(* Logix 5000 project; controller WWTP_SOLIDS_CLX vendor 1 type 14 code 54 rev 17.2; software revision 17.00; part 11 of 16 *)

ADD_ON_INSTRUCTION P_ResInh   (* revision 0.12, ExecutePrescan, ExecuteEnableInFalse *)
// Restart Inhibit
// Revision note:
// Aligned name, description and local STRING values, sizes, across instructions.
// Help:
// This Instruction monitors starts, running and stops of a motor and decides, based
// on rules for winding heating, when the motor can be started again.
// This Instruction uses a state model, which is documented in the User
// Documentation for the instruction.  It has the following states:
// *  S01:  Cold Motor Ready to Start
// *  S02:  Cold Motor Starting
// *  S03:  Cold Motor Running
// *  S04:  Cold Motor First Failure to Start
// *  S05:  Cold Motor Subsequent Failure to Start
// *  S06:  Hot Motor Starting
// *  S07:  Hot Motor Running
// *  S08:  Hot Motor Short Run Then Stopped
// *  S09:  Hot Motor Long Run Then Stopped
// *  S10:  Hot Motor First Failure to Start
// *  S11:  Hot Motor Subsequent Failure to Start
// *  S12:  Hot Motor Ready to Start
// NOTE:  This is a very basic state model for motor heating and is not intended
// as a close physical model of any given motor.  It cannot replace more
// extensive or sensor-based motor monitoring and modelling systems.
// NOTE:  EnableInFalse (false rung) is treated the same a motor stopped
// (Inp_Starting = 0, Inp_Running = 0, Inp_Stopped = 1).
VAR_INPUT
   Inp_Stopped : BOOL; {visible}   // Equipment is confirmed Stopped
   Inp_Starting : BOOL; {visible}   // Equipment is Starting, indicating a start attempt
   Inp_Running : BOOL := 1; {visible}   // Equipment is confirmed Running
   Cfg_ThreeColdStarts : DINT := 1800;   // Sec within which three starts are allowed if cold
   Cfg_FirstFailCold : DINT := 1800;   // Sec for cold motor to wait after 1st start failure before ready to start
   Cfg_SubseqFailCold : DINT := 14400;   // Sec for cold motor to wait after 2nd and subsequent start failure before ready
   Cfg_FirstFailHot : DINT := 1800;   // Sec for hot motor to wait after 1st start failure before ready to start
   Cfg_SubseqFailHot : DINT := 14400;   // Sec for hot motor to wait after 2nd and subsequent start failure before ready
   Cfg_HotRestartOK : DINT := 3600;   // Sec for hot motor to run so it can immediately restart after stop
   Cfg_RestartHot : DINT := 3600;   // Sec for hot motor to wait after stop if stopped before Hot Restart OK time
   Cfg_HotToCold : DINT := 57600;   // Sec for a stopped hot motor to become cold
END_VAR
VAR_OUTPUT
   Val_MinToReady : DINT; {visible}   // Minutes yet inhibited before ready to start (mmm:ss)
   Val_SecToReady : DINT; {visible}   // Seconds yet inhibited before ready to start (mmm:ss)
   Val_State : DINT := 1;   // State Number (see State Diagram in docs) for HMI
   Sts_Ready : BOOL; {visible}   // Permissive for unit to start 1=ready, 0=not ready
   Sts_Err : BOOL; {visible}   // 1=Error in Config: Invalid Time (use 0.0 to 2147483)
END_VAR
VAR
   Wrk_FirstColdStartT : TIMER := (PRE := 1800000);   // Time since first cold start
   Wrk_FirstFailColdT : TIMER := (PRE := 1800000);   // Time for cold motor to wait after 1st start failure before ready
   Wrk_SubsFailColdT : TIMER := (PRE := 14400000);   // Time for cold motor to wait after 2nd and subs. failures before ready
   Wrk_FirstFailHotT : TIMER := (PRE := 1800000);   // Time for hot motor to wait after 1st start failure before ready
   Wrk_SubsFailHotT : TIMER := (PRE := 14400000);   // Time for hot motor to wait after 2nd and subs. failures before ready
   Wrk_HotRestartOKT : TIMER := (PRE := 14400000);   // Time for hot motor to run so it can restart immediately when stopped
   Wrk_RestartHotT : TIMER := (PRE := 3600000);   // Time for hot motor to wait after stop after running less than Hot Restart OK time
   Wrk_HotToColdT : TIMER := (PRE := 57600000);   // Time for a stopped hot motor to become cold
   Wrk_FailCount : DINT;   // Number of failed start attempts
   Wrk_mSecUntilReady : DINT;   // Milliseconds until the inhibit time is done and the unit is ready to start
   Wrk_SecUntilReady : DINT;   // Seconds until inhibit time is done and the unit is ready to start
   Wrk_State : DINT := 1;   // Instruction State (see state diagram in design docs)
   Wrk_Ready : BOOL;   // Internal storage of Sts_Ready: 1 = OK to start
   Wrk_SecondColdStartT : TIMER := (PRE := 1800000);   // Time since second cold start
END_VAR

ROUTINE EnableInFalse   (* ladder *)
// Process state model for Motor as Not Running
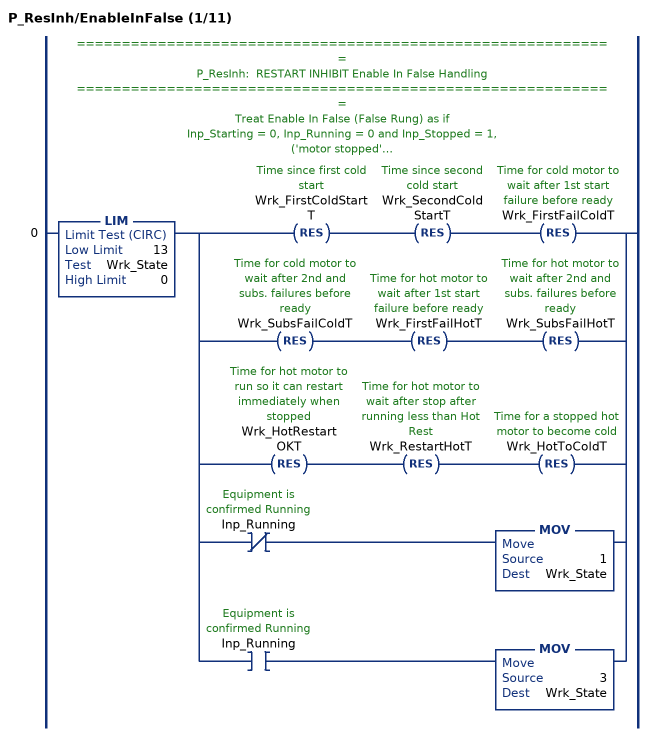
   // ============================================================
   // P_ResInh:  RESTART INHIBIT Enable In False Handling
   // ============================================================
   // Treat Enable In False (False Rung) as if
   //  Inp_Starting = 0, Inp_Running = 0 and Inp_Stopped = 1,
   // ('motor stopped')
   // This logic is identical to the main Logic Routine except that actions with the Motor
   // Running or Starting have been removed, and all actions with the Motor
   // Stopped have been made unconditional.  Adjacent unconditional rungs
   // have been combined to save memory.
   // ============================================================
   // INVALID STATE
   // ============================================================
   // If the State number is not valid (valid states are 1..12),
   //  the various timers are reset (all are retentive), and the State Machine is set to:
   // *  State S01  ( Cold Motor Ready to Start )  if the pump is NOT Running, or
   // *  State S03  ( Cold Motor Running )  if the pump is Running.
   0: LIM(13,Wrk_State,0)[RES(Wrk_FirstColdStartT) RES(Wrk_SecondColdStartT) RES(Wrk_FirstFailColdT) ,RES(Wrk_SubsFailColdT) RES(Wrk_FirstFailHotT) RES(Wrk_SubsFailHotT) ,RES(Wrk_HotRestartOKT) RES(Wrk_RestartHotT) RES(Wrk_HotToColdT) ,XIO(Inp_Running) MOV(1,Wrk_State) ,XIC(Inp_Running) MOV(3,Wrk_State) ];
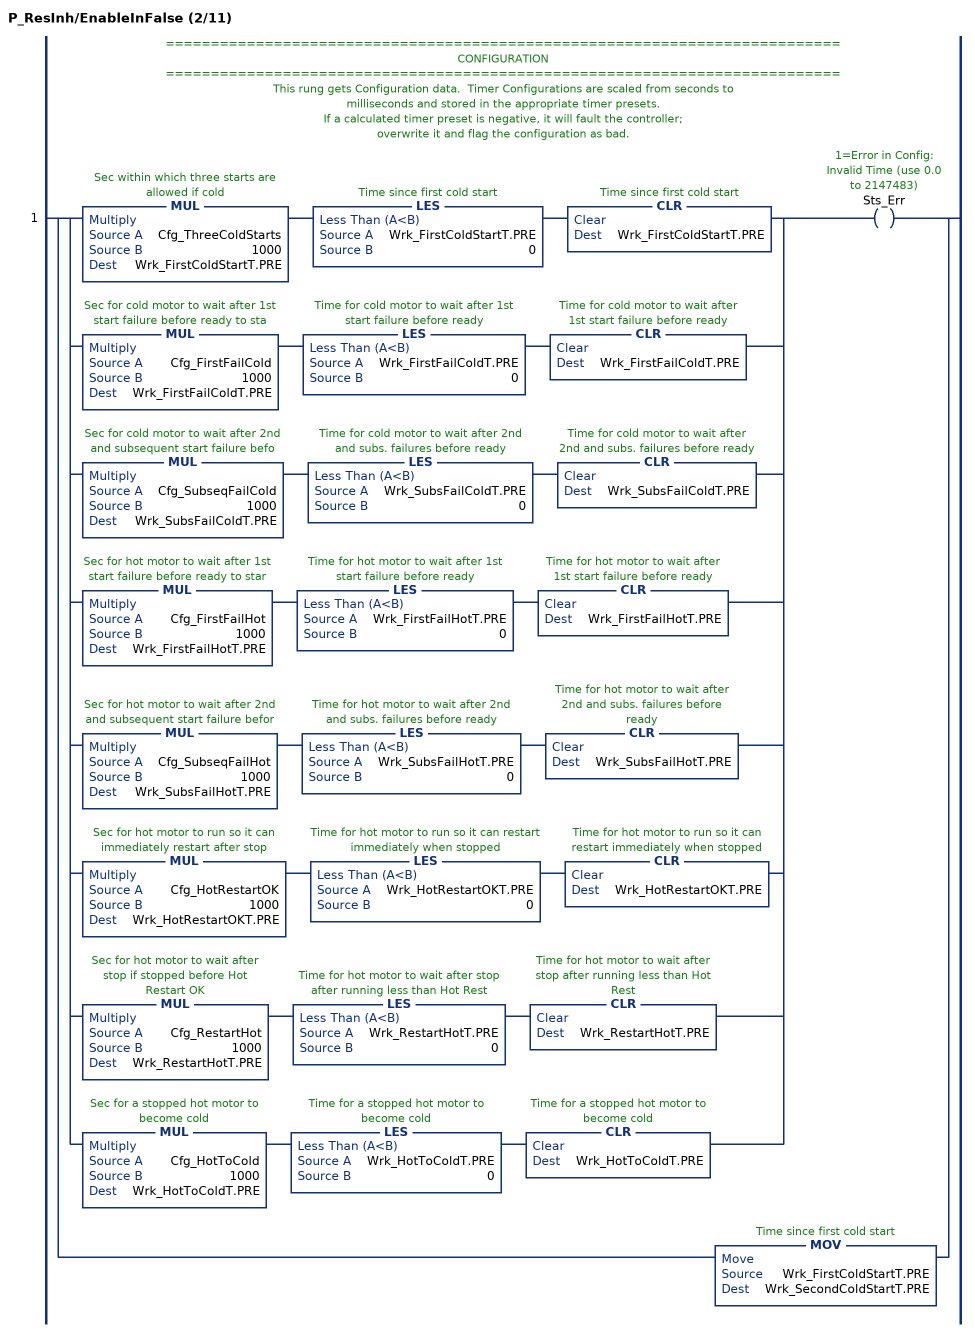
   // ===========================================================================
   // CONFIGURATION
   // ===========================================================================
   // This rung gets Configuration data.  Timer Configurations are scaled from seconds to
   // milliseconds and stored in the appropriate timer presets.
   // If a calculated timer preset is negative, it will fault the controller;
   // overwrite it and flag the configuration as bad.
   1: [[MUL(Cfg_ThreeColdStarts,1000,Wrk_FirstColdStartT.PRE) LES(Wrk_FirstColdStartT.PRE,0) CLR(Wrk_FirstColdStartT.PRE) ,MUL(Cfg_FirstFailCold,1000,Wrk_FirstFailColdT.PRE) LES(Wrk_FirstFailColdT.PRE,0) CLR(Wrk_FirstFailColdT.PRE) ,MUL(Cfg_SubseqFailCold,1000,Wrk_SubsFailColdT.PRE) LES(Wrk_SubsFailColdT.PRE,0) CLR(Wrk_SubsFailColdT.PRE) ,MUL(Cfg_FirstFailHot,1000,Wrk_FirstFailHotT.PRE) LES(Wrk_FirstFailHotT.PRE,0) CLR(Wrk_FirstFailHotT.PRE) ,MUL(Cfg_SubseqFailHot,1000,Wrk_SubsFailHotT.PRE) LES(Wrk_SubsFailHotT.PRE,0) CLR(Wrk_SubsFailHotT.PRE) ,MUL(Cfg_HotRestartOK,1000,Wrk_HotRestartOKT.PRE) LES(Wrk_HotRestartOKT.PRE,0) CLR(Wrk_HotRestartOKT.PRE) ,MUL(Cfg_RestartHot,1000,Wrk_RestartHotT.PRE) LES(Wrk_RestartHotT.PRE,0) CLR(Wrk_RestartHotT.PRE) ,MUL(Cfg_HotToCold,1000,Wrk_HotToColdT.PRE) LES(Wrk_HotToColdT.PRE,0) CLR(Wrk_HotToColdT.PRE) ] OTE(Sts_Err) ,MOV(Wrk_FirstColdStartT.PRE,Wrk_SecondColdStartT.PRE) ];
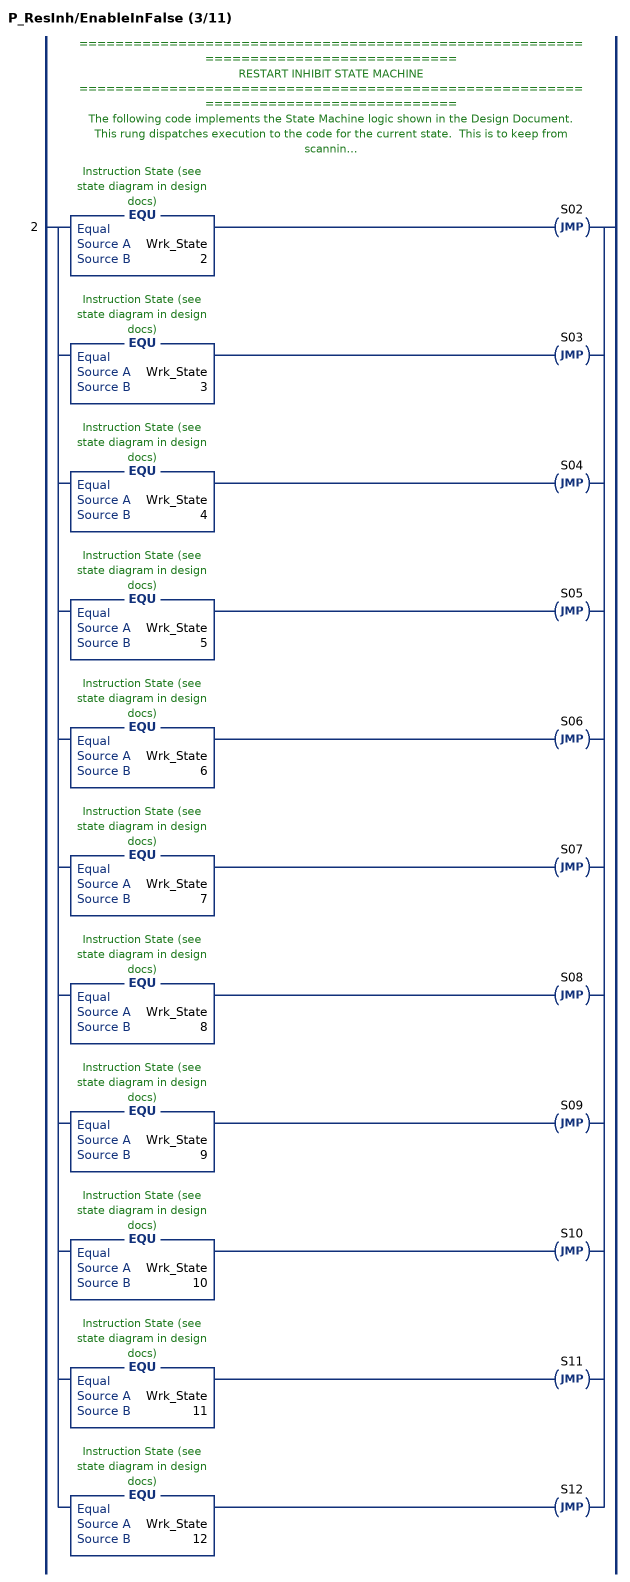
   // ====================================================================================
   // RESTART INHIBIT STATE MACHINE
   // ====================================================================================
   // The following code implements the State Machine logic shown in the Design Document.
   // This rung dispatches execution to the code for the current state.  This is to keep from scanning
   // the code for all the states every scan, and so that certain timers can be shared by multiple states.
   // (For State = 1, execution just falls through into the State 1 code.)
   2: [EQU(Wrk_State,2) JMP(S02) ,EQU(Wrk_State,3) JMP(S03) ,EQU(Wrk_State,4) JMP(S04) ,EQU(Wrk_State,5) JMP(S05) ,EQU(Wrk_State,6) JMP(S06) ,EQU(Wrk_State,7) JMP(S07) ,EQU(Wrk_State,8) JMP(S08) ,EQU(Wrk_State,9) JMP(S09) ,EQU(Wrk_State,10) JMP(S10) ,EQU(Wrk_State,11) JMP(S11) ,EQU(Wrk_State,12) JMP(S12) ];
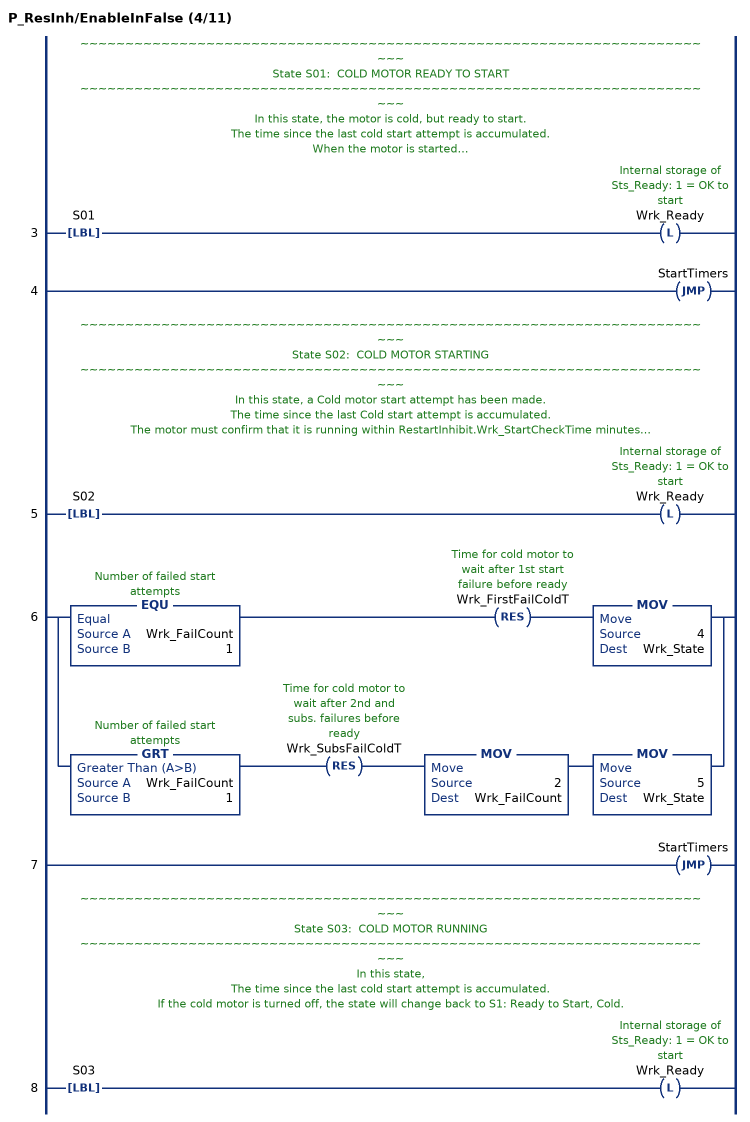
   // ~~~~~~~~~~~~~~~~~~~~~~~~~~~~~~~~~~~~~~~~~~~~~~~~~~~~~~~~~~~~~~~~~~~~~~~~
   // State S01:  COLD MOTOR READY TO START
   // ~~~~~~~~~~~~~~~~~~~~~~~~~~~~~~~~~~~~~~~~~~~~~~~~~~~~~~~~~~~~~~~~~~~~~~~~
   // In this state, the motor is cold, but ready to start.
   // The time since the last cold start attempt is accumulated.
   // When the motor is started:
   // If it has been at least Last Cold Start minutes since the last attempt was made to start the motor,
   // the motor is still considered cold, it has had enough time to cool off.
   // If it has been less than Last Cold Start minutes since the last attempt was made to start the motor,
   // the motor is considered hot due to multiple re-starts in too short a time period.
   3: LBL(S01)OTL(Wrk_Ready);
   4: JMP(StartTimers);
   // ~~~~~~~~~~~~~~~~~~~~~~~~~~~~~~~~~~~~~~~~~~~~~~~~~~~~~~~~~~~~~~~~~~~~~~~~
   // State S02:  COLD MOTOR STARTING
   // ~~~~~~~~~~~~~~~~~~~~~~~~~~~~~~~~~~~~~~~~~~~~~~~~~~~~~~~~~~~~~~~~~~~~~~~~
   // In this state, a Cold motor start attempt has been made.
   // The time since the last Cold start attempt is accumulated.
   // The motor must confirm that it is running within RestartInhibit.Wrk_StartCheckTime minutes.
   // If it does, the state will change to S3: Cold Motor Running
   // If it does not start properly within the allowable time, the state will change to either S4: 1st Failed Cold Restart, or S5: Subsequent Cold Failed Restart.
   5: LBL(S02)OTL(Wrk_Ready);
   6: [EQU(Wrk_FailCount,1) RES(Wrk_FirstFailColdT) MOV(4,Wrk_State) ,GRT(Wrk_FailCount,1) RES(Wrk_SubsFailColdT) MOV(2,Wrk_FailCount) MOV(5,Wrk_State) ];
   7: JMP(StartTimers);
   // ~~~~~~~~~~~~~~~~~~~~~~~~~~~~~~~~~~~~~~~~~~~~~~~~~~~~~~~~~~~~~~~~~~~~~~~~
   // State S03:  COLD MOTOR RUNNING
   // ~~~~~~~~~~~~~~~~~~~~~~~~~~~~~~~~~~~~~~~~~~~~~~~~~~~~~~~~~~~~~~~~~~~~~~~~
   // In this state,
   // The time since the last cold start attempt is accumulated.
   // If the cold motor is turned off, the state will change back to S1: Ready to Start, Cold.
   8: LBL(S03)OTL(Wrk_Ready);
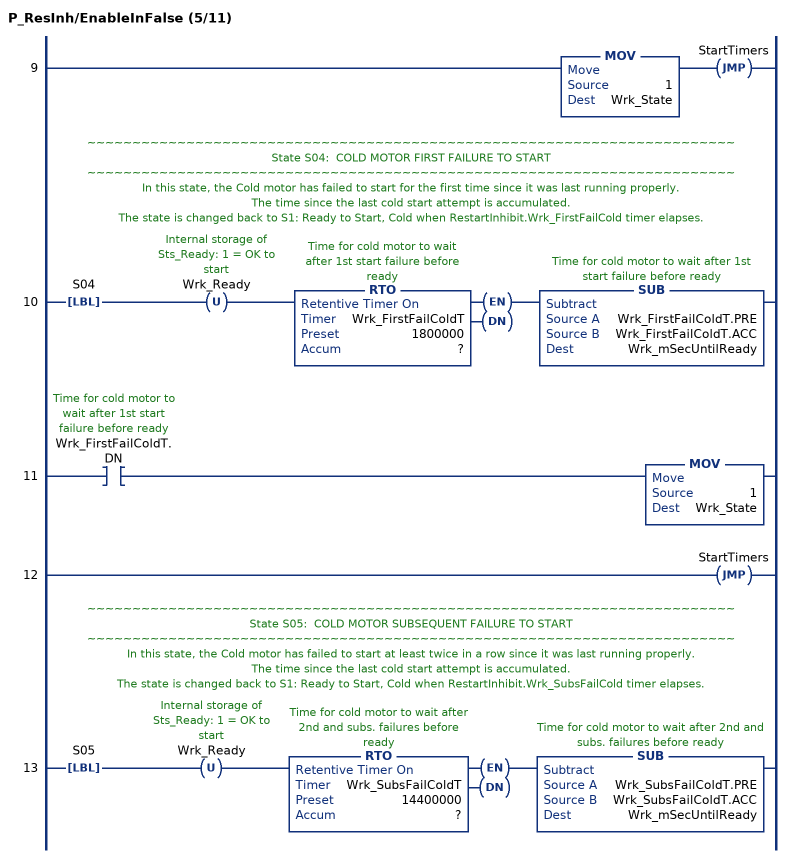
   9: MOV(1,Wrk_State)JMP(StartTimers);
   // ~~~~~~~~~~~~~~~~~~~~~~~~~~~~~~~~~~~~~~~~~~~~~~~~~~~~~~~~~~~~~~~~~~~~~~~~
   // State S04:  COLD MOTOR FIRST FAILURE TO START
   // ~~~~~~~~~~~~~~~~~~~~~~~~~~~~~~~~~~~~~~~~~~~~~~~~~~~~~~~~~~~~~~~~~~~~~~~~
   // In this state, the Cold motor has failed to start for the first time since it was last running properly.
   // The time since the last cold start attempt is accumulated.
   // The state is changed back to S1: Ready to Start, Cold when RestartInhibit.Wrk_FirstFailCold timer elapses.
   10: LBL(S04)OTU(Wrk_Ready)RTO(Wrk_FirstFailColdT,?,?)SUB(Wrk_FirstFailColdT.PRE,Wrk_FirstFailColdT.ACC,Wrk_mSecUntilReady);
   11: XIC(Wrk_FirstFailColdT.DN)MOV(1,Wrk_State);
   12: JMP(StartTimers);
   // ~~~~~~~~~~~~~~~~~~~~~~~~~~~~~~~~~~~~~~~~~~~~~~~~~~~~~~~~~~~~~~~~~~~~~~~~
   // State S05:  COLD MOTOR SUBSEQUENT FAILURE TO START
   // ~~~~~~~~~~~~~~~~~~~~~~~~~~~~~~~~~~~~~~~~~~~~~~~~~~~~~~~~~~~~~~~~~~~~~~~~
   // In this state, the Cold motor has failed to start at least twice in a row since it was last running properly.
   // The time since the last cold start attempt is accumulated.
   // The state is changed back to S1: Ready to Start, Cold when RestartInhibit.Wrk_SubsFailCold timer elapses.
   13: LBL(S05)OTU(Wrk_Ready)RTO(Wrk_SubsFailColdT,?,?)SUB(Wrk_SubsFailColdT.PRE,Wrk_SubsFailColdT.ACC,Wrk_mSecUntilReady);
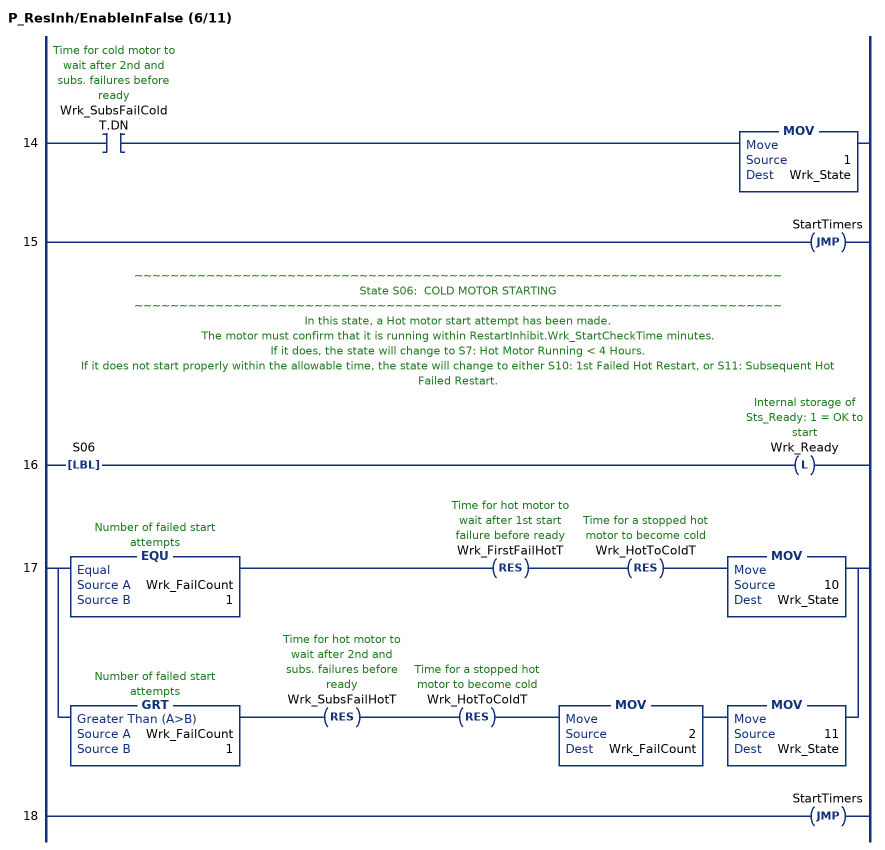
   14: XIC(Wrk_SubsFailColdT.DN)MOV(1,Wrk_State);
   15: JMP(StartTimers);
   // ~~~~~~~~~~~~~~~~~~~~~~~~~~~~~~~~~~~~~~~~~~~~~~~~~~~~~~~~~~~~~~~~~~~~~~~~
   // State S06:  COLD MOTOR STARTING
   // ~~~~~~~~~~~~~~~~~~~~~~~~~~~~~~~~~~~~~~~~~~~~~~~~~~~~~~~~~~~~~~~~~~~~~~~~
   // In this state, a Hot motor start attempt has been made.
   // The motor must confirm that it is running within RestartInhibit.Wrk_StartCheckTime minutes.
   // If it does, the state will change to S7: Hot Motor Running < 4 Hours.
   // If it does not start properly within the allowable time, the state will change to either S10: 1st Failed Hot Restart, or S11: Subsequent Hot Failed Restart.
   16: LBL(S06)OTL(Wrk_Ready);
   17: [EQU(Wrk_FailCount,1) RES(Wrk_FirstFailHotT) RES(Wrk_HotToColdT) MOV(10,Wrk_State) ,GRT(Wrk_FailCount,1) RES(Wrk_SubsFailHotT) RES(Wrk_HotToColdT) MOV(2,Wrk_FailCount) MOV(11,Wrk_State) ];
   18: JMP(StartTimers);
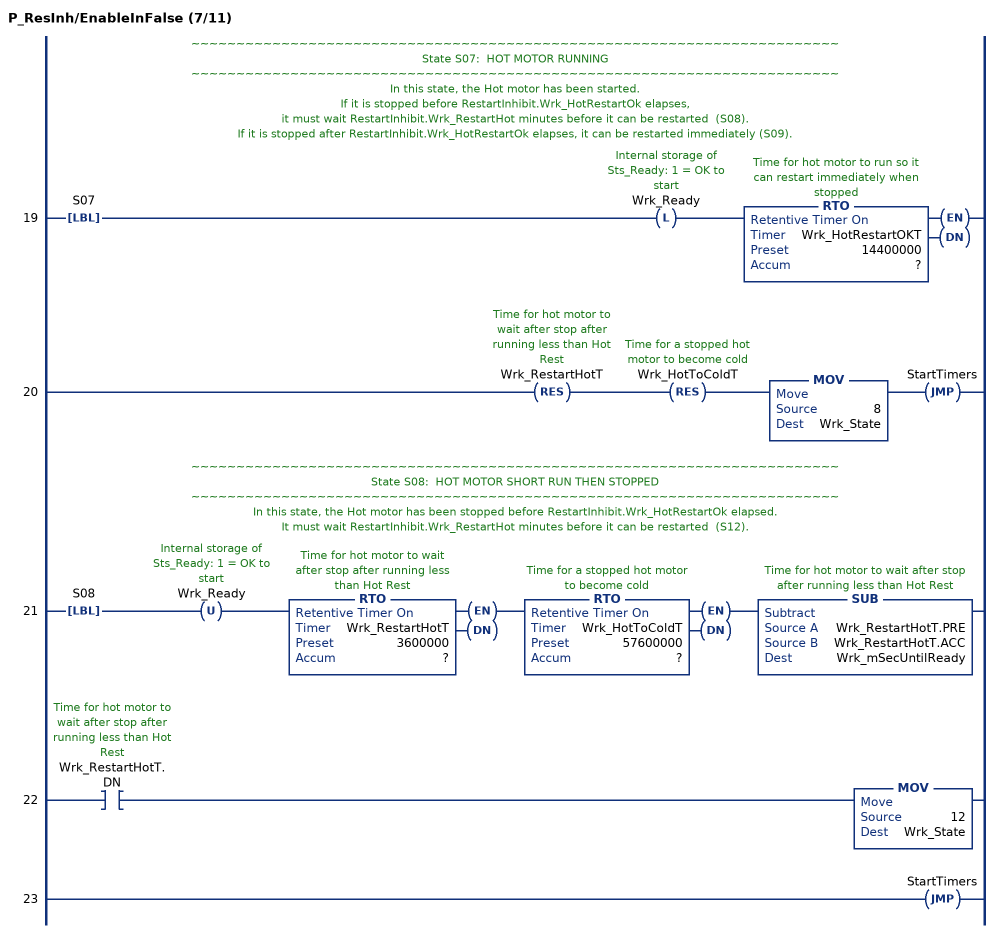
   // ~~~~~~~~~~~~~~~~~~~~~~~~~~~~~~~~~~~~~~~~~~~~~~~~~~~~~~~~~~~~~~~~~~~~~~~~
   // State S07:  HOT MOTOR RUNNING
   // ~~~~~~~~~~~~~~~~~~~~~~~~~~~~~~~~~~~~~~~~~~~~~~~~~~~~~~~~~~~~~~~~~~~~~~~~
   // In this state, the Hot motor has been started.
   // If it is stopped before RestartInhibit.Wrk_HotRestartOk elapses,
   // it must wait RestartInhibit.Wrk_RestartHot minutes before it can be restarted  (S08).
   // If it is stopped after RestartInhibit.Wrk_HotRestartOk elapses, it can be restarted immediately (S09).
   19: LBL(S07)OTL(Wrk_Ready)RTO(Wrk_HotRestartOKT,?,?);
   20: RES(Wrk_RestartHotT)RES(Wrk_HotToColdT)MOV(8,Wrk_State)JMP(StartTimers);
   // ~~~~~~~~~~~~~~~~~~~~~~~~~~~~~~~~~~~~~~~~~~~~~~~~~~~~~~~~~~~~~~~~~~~~~~~~
   // State S08:  HOT MOTOR SHORT RUN THEN STOPPED
   // ~~~~~~~~~~~~~~~~~~~~~~~~~~~~~~~~~~~~~~~~~~~~~~~~~~~~~~~~~~~~~~~~~~~~~~~~
   // In this state, the Hot motor has been stopped before RestartInhibit.Wrk_HotRestartOk elapsed.
   // It must wait RestartInhibit.Wrk_RestartHot minutes before it can be restarted  (S12).
   21: LBL(S08)OTU(Wrk_Ready)RTO(Wrk_RestartHotT,?,?)RTO(Wrk_HotToColdT,?,?)SUB(Wrk_RestartHotT.PRE,Wrk_RestartHotT.ACC,Wrk_mSecUntilReady);
   22: XIC(Wrk_RestartHotT.DN)MOV(12,Wrk_State);
   23: JMP(StartTimers);
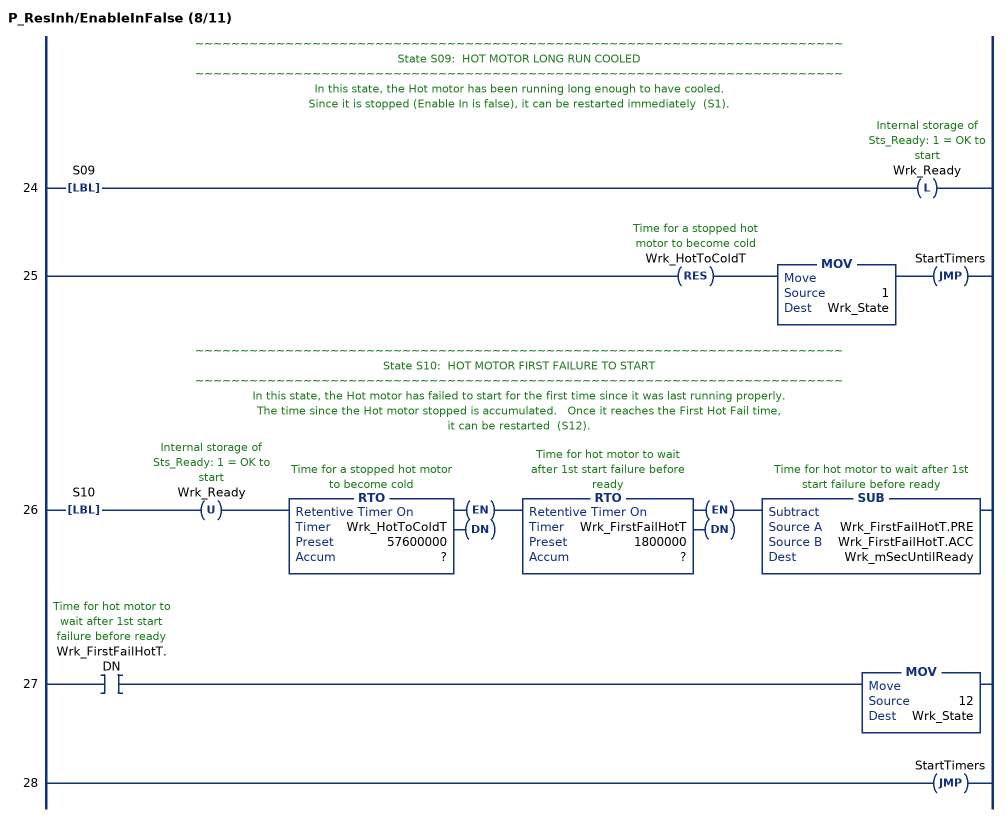
   // ~~~~~~~~~~~~~~~~~~~~~~~~~~~~~~~~~~~~~~~~~~~~~~~~~~~~~~~~~~~~~~~~~~~~~~~~
   // State S09:  HOT MOTOR LONG RUN COOLED
   // ~~~~~~~~~~~~~~~~~~~~~~~~~~~~~~~~~~~~~~~~~~~~~~~~~~~~~~~~~~~~~~~~~~~~~~~~
   // In this state, the Hot motor has been running long enough to have cooled.
   // Since it is stopped (Enable In is false), it can be restarted immediately  (S1).
   24: LBL(S09)OTL(Wrk_Ready);
   25: RES(Wrk_HotToColdT)MOV(1,Wrk_State)JMP(StartTimers);
   // ~~~~~~~~~~~~~~~~~~~~~~~~~~~~~~~~~~~~~~~~~~~~~~~~~~~~~~~~~~~~~~~~~~~~~~~~
   // State S10:  HOT MOTOR FIRST FAILURE TO START
   // ~~~~~~~~~~~~~~~~~~~~~~~~~~~~~~~~~~~~~~~~~~~~~~~~~~~~~~~~~~~~~~~~~~~~~~~~
   // In this state, the Hot motor has failed to start for the first time since it was last running properly.
   // The time since the Hot motor stopped is accumulated.   Once it reaches the First Hot Fail time,
   // it can be restarted  (S12).
   26: LBL(S10)OTU(Wrk_Ready)RTO(Wrk_HotToColdT,?,?)RTO(Wrk_FirstFailHotT,?,?)SUB(Wrk_FirstFailHotT.PRE,Wrk_FirstFailHotT.ACC,Wrk_mSecUntilReady);
   27: XIC(Wrk_FirstFailHotT.DN)MOV(12,Wrk_State);
   28: JMP(StartTimers);
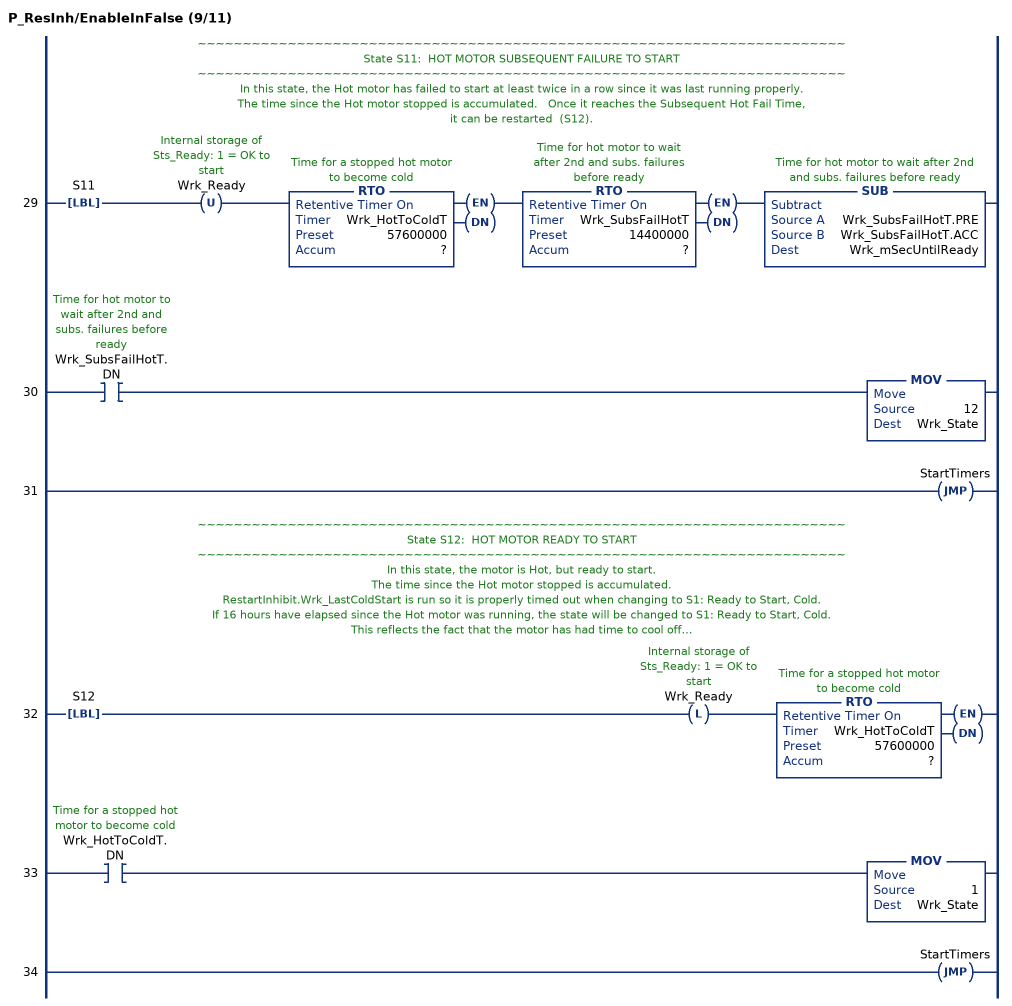
   // ~~~~~~~~~~~~~~~~~~~~~~~~~~~~~~~~~~~~~~~~~~~~~~~~~~~~~~~~~~~~~~~~~~~~~~~~
   // State S11:  HOT MOTOR SUBSEQUENT FAILURE TO START
   // ~~~~~~~~~~~~~~~~~~~~~~~~~~~~~~~~~~~~~~~~~~~~~~~~~~~~~~~~~~~~~~~~~~~~~~~~
   // In this state, the Hot motor has failed to start at least twice in a row since it was last running properly.
   // The time since the Hot motor stopped is accumulated.   Once it reaches the Subsequent Hot Fail Time,
   // it can be restarted  (S12).
   29: LBL(S11)OTU(Wrk_Ready)RTO(Wrk_HotToColdT,?,?)RTO(Wrk_SubsFailHotT,?,?)SUB(Wrk_SubsFailHotT.PRE,Wrk_SubsFailHotT.ACC,Wrk_mSecUntilReady);
   30: XIC(Wrk_SubsFailHotT.DN)MOV(12,Wrk_State);
   31: JMP(StartTimers);
   // ~~~~~~~~~~~~~~~~~~~~~~~~~~~~~~~~~~~~~~~~~~~~~~~~~~~~~~~~~~~~~~~~~~~~~~~~
   // State S12:  HOT MOTOR READY TO START
   // ~~~~~~~~~~~~~~~~~~~~~~~~~~~~~~~~~~~~~~~~~~~~~~~~~~~~~~~~~~~~~~~~~~~~~~~~
   // In this state, the motor is Hot, but ready to start.
   // The time since the Hot motor stopped is accumulated.
   // RestartInhibit.Wrk_LastColdStart is run so it is properly timed out when changing to S1: Ready to Start, Cold.
   // If 16 hours have elapsed since the Hot motor was running, the state will be changed to S1: Ready to Start, Cold.
   // This reflects the fact that the motor has had time to cool off.
   // Otherwise, the logic waits for a Start attempt to change the state to S6: Start Check, Hot.
   32: LBL(S12)OTL(Wrk_Ready)RTO(Wrk_HotToColdT,?,?);
   33: XIC(Wrk_HotToColdT.DN)MOV(1,Wrk_State);
   34: JMP(StartTimers);
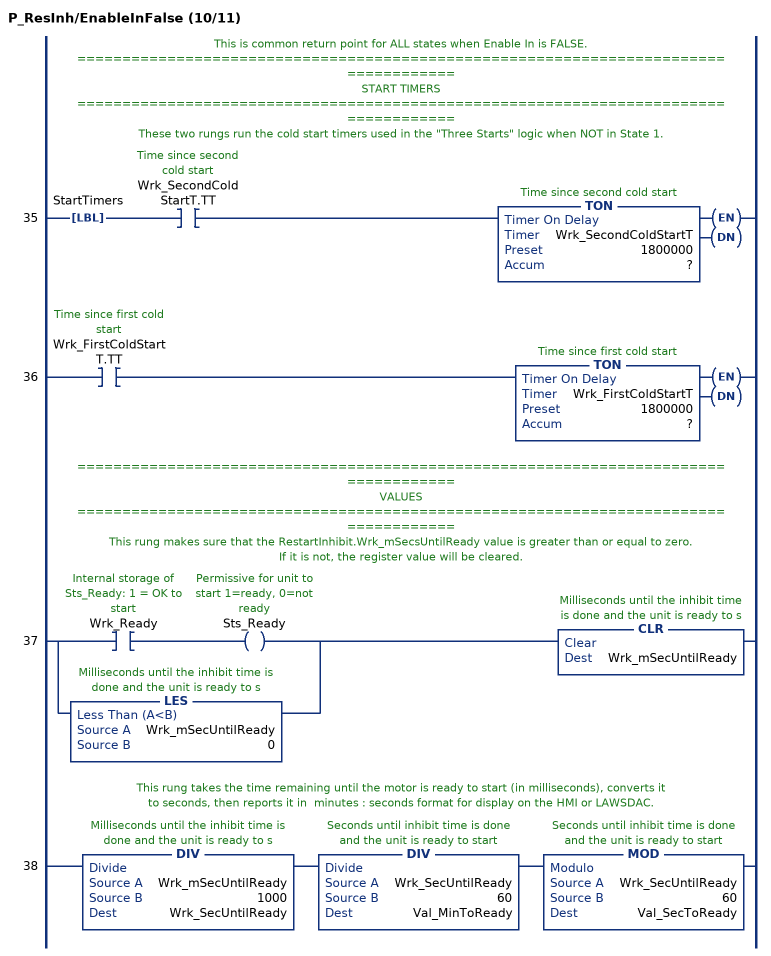
   // This is common return point for ALL states when Enable In is FALSE.
   // ====================================================================================
   // START TIMERS
   // ====================================================================================
   // These two rungs run the cold start timers used in the "Three Starts" logic when NOT in State 1.
   35: LBL(StartTimers)XIC(Wrk_SecondColdStartT.TT)TON(Wrk_SecondColdStartT,?,?);
   36: XIC(Wrk_FirstColdStartT.TT)TON(Wrk_FirstColdStartT,?,?);
   // ====================================================================================
   // VALUES
   // ====================================================================================
   // This rung makes sure that the RestartInhibit.Wrk_mSecsUntilReady value is greater than or equal to zero.
   // If it is not, the register value will be cleared.
   37: [XIC(Wrk_Ready) OTE(Sts_Ready) ,LES(Wrk_mSecUntilReady,0) ]CLR(Wrk_mSecUntilReady);
   // This rung takes the time remaining until the motor is ready to start (in milliseconds), converts it
   // to seconds, then reports it in  minutes : seconds format for display on the HMI or LAWSDAC.
   38: DIV(Wrk_mSecUntilReady,1000,Wrk_SecUntilReady)DIV(Wrk_SecUntilReady,60,Val_MinToReady)MOD(Wrk_SecUntilReady,60,Val_SecToReady);
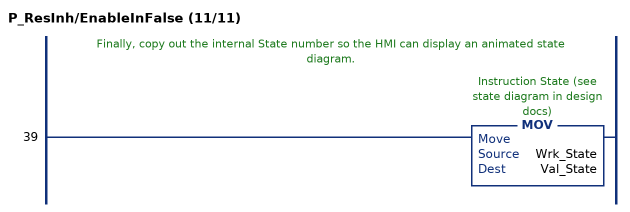
   // Finally, copy out the internal State number so the HMI can display an animated state diagram.
   39: MOV(Wrk_State,Val_State);
END_ROUTINE

ROUTINE Logic   (* ladder *)
// Determine motor readiness based on restart rules
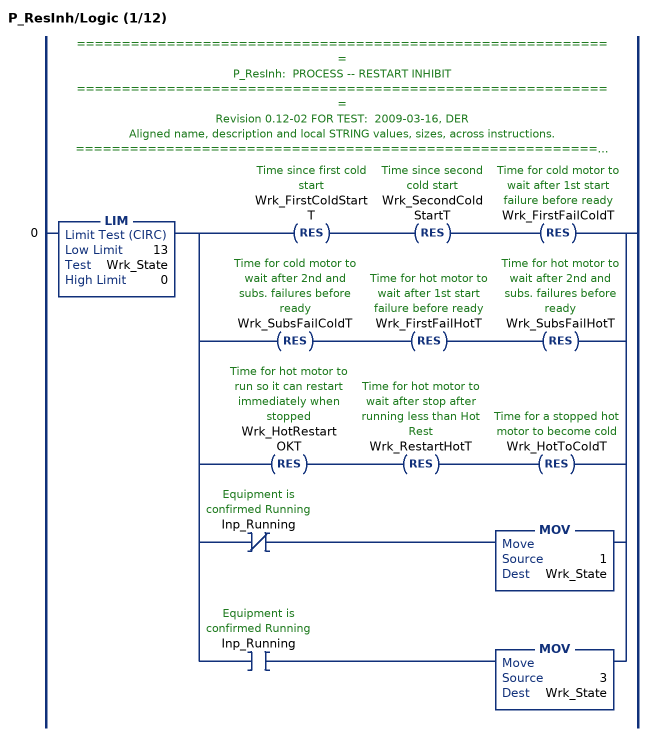
   // ============================================================
   // P_ResInh:  PROCESS -- RESTART INHIBIT
   // ============================================================
   // Revision 0.12-02 FOR TEST:  2009-03-16, DER
   // Aligned name, description and local STRING values, sizes, across instructions.
   // ============================================================
   // This Instruction monitors starts, running and stops of a motor and decides, based on
   // simple criteria for winding heating, when the motor can be started again.
   // This Instruction is largely State Machine-based.  It has the following states:
   // *  S01:  Cold Motor Ready to Start
   // *  S02:  Cold Motor Starting
   // *  S03:  Cold Motor Running
   // *  S04:  Cold Motor First Failure to Start
   // *  S05:  Cold Motor Subsequent Failure to Start
   // *  S06:  Hot Motor Starting
   // *  S07:  Hot Motor Running
   // *  S08:  Hot Motor Short Run Then Stopped
   // *  S09:  Hot Motor Long Run Cooled
   // *  S10:  Hot Motor First Failure to Start
   // *  S11:  Hot Motor Subsequent Failure to Start
   // *  S12:  Hot Motor Ready to Start
   // Refer to the state diagram in the End User Documentation for details.
   // NOTE: The state is stored in a Local Tag and not available outside to other
   // instructions, but can be shown on an HMI.
   // ============================================================
   // INVALID STATE
   // ============================================================
   // If the State number is not valid (valid states are 1..12),
   //  the various timers are reset (all are retentive), and the State Machine is set to:
   // *  State S01  ( Cold Motor Ready to Start )  if the pump is NOT Running, or
   // *  State S03  ( Cold Motor Running )  if the pump is Running.
   0: LIM(13,Wrk_State,0)[RES(Wrk_FirstColdStartT) RES(Wrk_SecondColdStartT) RES(Wrk_FirstFailColdT) ,RES(Wrk_SubsFailColdT) RES(Wrk_FirstFailHotT) RES(Wrk_SubsFailHotT) ,RES(Wrk_HotRestartOKT) RES(Wrk_RestartHotT) RES(Wrk_HotToColdT) ,XIO(Inp_Running) MOV(1,Wrk_State) ,XIC(Inp_Running) MOV(3,Wrk_State) ];
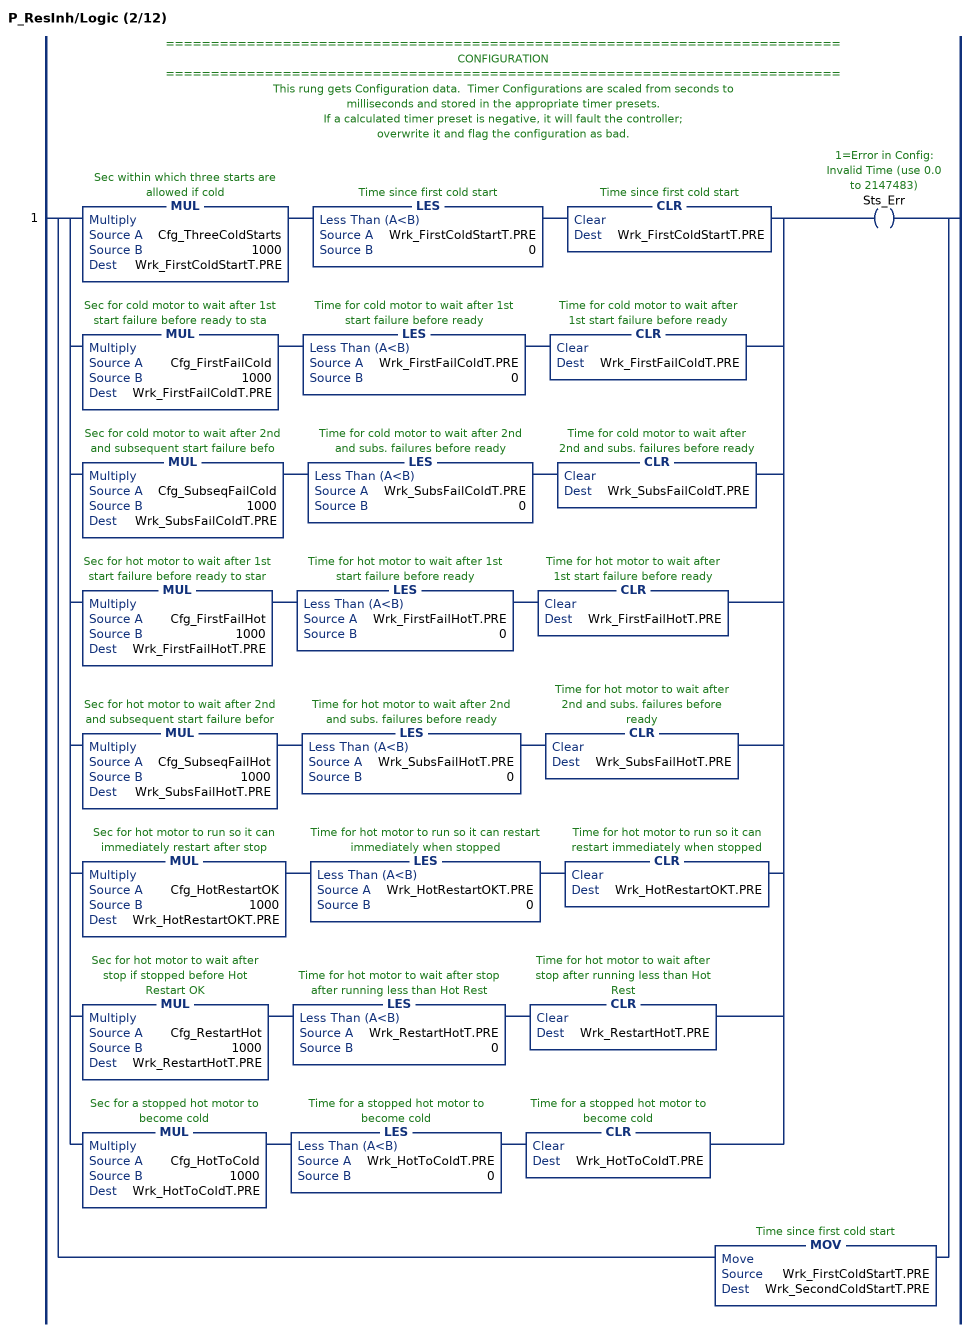
   // ===========================================================================
   // CONFIGURATION
   // ===========================================================================
   // This rung gets Configuration data.  Timer Configurations are scaled from seconds to
   // milliseconds and stored in the appropriate timer presets.
   // If a calculated timer preset is negative, it will fault the controller;
   // overwrite it and flag the configuration as bad.
   1: [[MUL(Cfg_ThreeColdStarts,1000,Wrk_FirstColdStartT.PRE) LES(Wrk_FirstColdStartT.PRE,0) CLR(Wrk_FirstColdStartT.PRE) ,MUL(Cfg_FirstFailCold,1000,Wrk_FirstFailColdT.PRE) LES(Wrk_FirstFailColdT.PRE,0) CLR(Wrk_FirstFailColdT.PRE) ,MUL(Cfg_SubseqFailCold,1000,Wrk_SubsFailColdT.PRE) LES(Wrk_SubsFailColdT.PRE,0) CLR(Wrk_SubsFailColdT.PRE) ,MUL(Cfg_FirstFailHot,1000,Wrk_FirstFailHotT.PRE) LES(Wrk_FirstFailHotT.PRE,0) CLR(Wrk_FirstFailHotT.PRE) ,MUL(Cfg_SubseqFailHot,1000,Wrk_SubsFailHotT.PRE) LES(Wrk_SubsFailHotT.PRE,0) CLR(Wrk_SubsFailHotT.PRE) ,MUL(Cfg_HotRestartOK,1000,Wrk_HotRestartOKT.PRE) LES(Wrk_HotRestartOKT.PRE,0) CLR(Wrk_HotRestartOKT.PRE) ,MUL(Cfg_RestartHot,1000,Wrk_RestartHotT.PRE) LES(Wrk_RestartHotT.PRE,0) CLR(Wrk_RestartHotT.PRE) ,MUL(Cfg_HotToCold,1000,Wrk_HotToColdT.PRE) LES(Wrk_HotToColdT.PRE,0) CLR(Wrk_HotToColdT.PRE) ] OTE(Sts_Err) ,MOV(Wrk_FirstColdStartT.PRE,Wrk_SecondColdStartT.PRE) ];
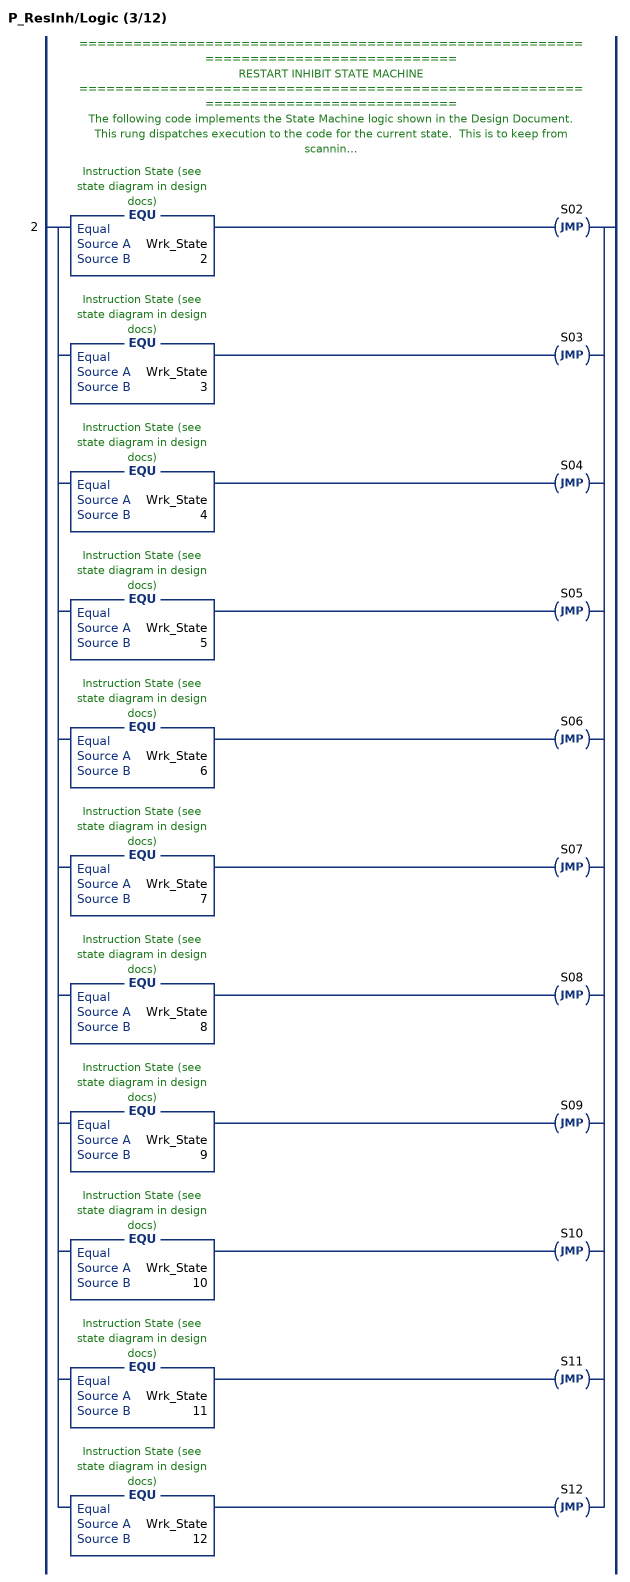
   // ====================================================================================
   // RESTART INHIBIT STATE MACHINE
   // ====================================================================================
   // The following code implements the State Machine logic shown in the Design Document.
   // This rung dispatches execution to the code for the current state.  This is to keep from scanning
   // the code for all the states every scan, and so that certain timers can be shared by multiple states.
   // (For State = 1, execution just falls through into the State 1 code.)
   2: [EQU(Wrk_State,2) JMP(S02) ,EQU(Wrk_State,3) JMP(S03) ,EQU(Wrk_State,4) JMP(S04) ,EQU(Wrk_State,5) JMP(S05) ,EQU(Wrk_State,6) JMP(S06) ,EQU(Wrk_State,7) JMP(S07) ,EQU(Wrk_State,8) JMP(S08) ,EQU(Wrk_State,9) JMP(S09) ,EQU(Wrk_State,10) JMP(S10) ,EQU(Wrk_State,11) JMP(S11) ,EQU(Wrk_State,12) JMP(S12) ];
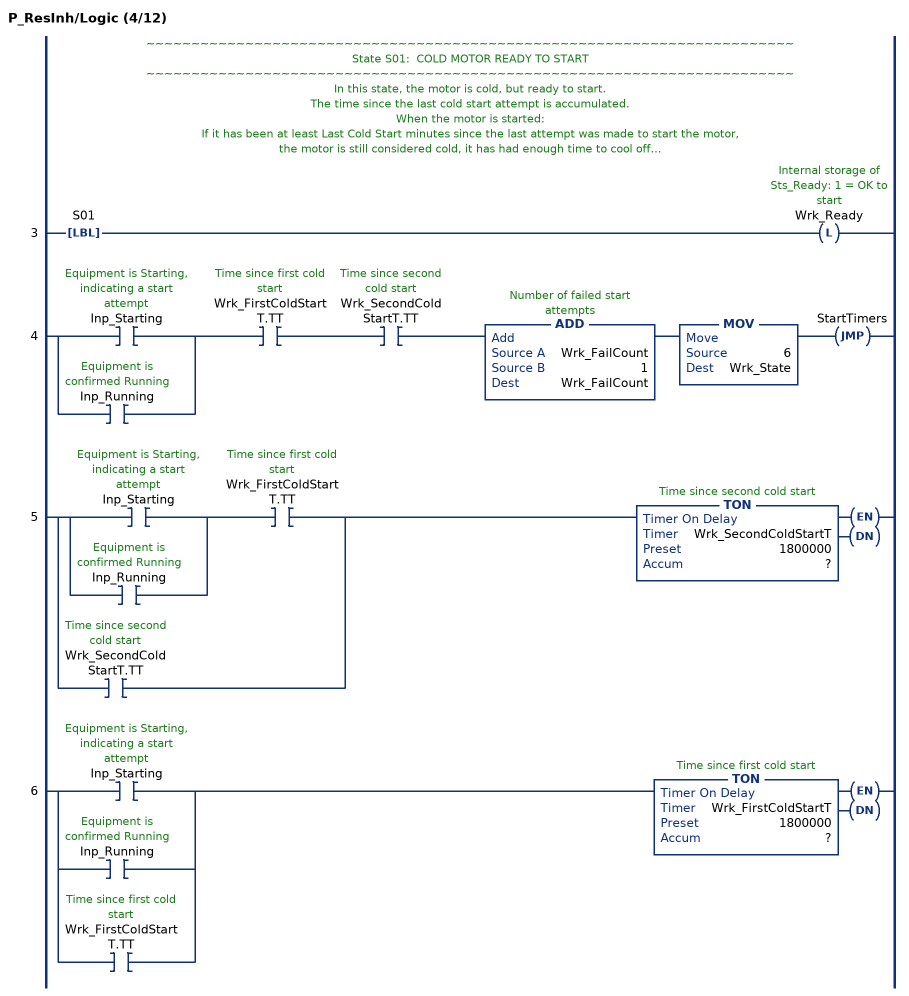
   // ~~~~~~~~~~~~~~~~~~~~~~~~~~~~~~~~~~~~~~~~~~~~~~~~~~~~~~~~~~~~~~~~~~~~~~~~
   // State S01:  COLD MOTOR READY TO START
   // ~~~~~~~~~~~~~~~~~~~~~~~~~~~~~~~~~~~~~~~~~~~~~~~~~~~~~~~~~~~~~~~~~~~~~~~~
   // In this state, the motor is cold, but ready to start.
   // The time since the last cold start attempt is accumulated.
   // When the motor is started:
   // If it has been at least Last Cold Start minutes since the last attempt was made to start the motor,
   // the motor is still considered cold, it has had enough time to cool off.
   // If it has been less than Last Cold Start minutes since the last attempt was made to start the motor,
   // the motor is considered hot due to multiple re-starts in too short a time period.
   3: LBL(S01)OTL(Wrk_Ready);
   4: [XIC(Inp_Starting) ,XIC(Inp_Running) ]XIC(Wrk_FirstColdStartT.TT)XIC(Wrk_SecondColdStartT.TT)ADD(Wrk_FailCount,1,Wrk_FailCount)MOV(6,Wrk_State)JMP(StartTimers);
   5: [[XIC(Inp_Starting) ,XIC(Inp_Running) ] XIC(Wrk_FirstColdStartT.TT) ,XIC(Wrk_SecondColdStartT.TT) ]TON(Wrk_SecondColdStartT,?,?);
   6: [[XIC(Inp_Starting) ,XIC(Inp_Running) ] ,XIC(Wrk_FirstColdStartT.TT) ]TON(Wrk_FirstColdStartT,?,?);
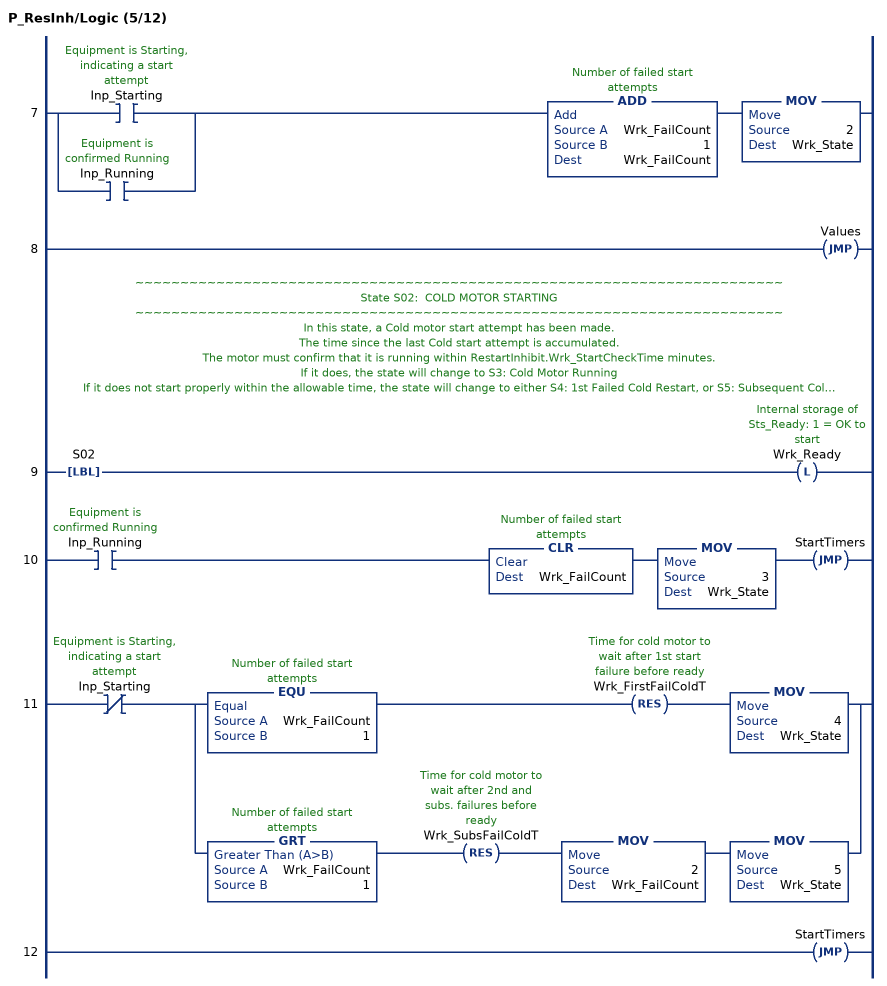
   7: [XIC(Inp_Starting) ,XIC(Inp_Running) ]ADD(Wrk_FailCount,1,Wrk_FailCount)MOV(2,Wrk_State);
   8: JMP(Values);
   // ~~~~~~~~~~~~~~~~~~~~~~~~~~~~~~~~~~~~~~~~~~~~~~~~~~~~~~~~~~~~~~~~~~~~~~~~
   // State S02:  COLD MOTOR STARTING
   // ~~~~~~~~~~~~~~~~~~~~~~~~~~~~~~~~~~~~~~~~~~~~~~~~~~~~~~~~~~~~~~~~~~~~~~~~
   // In this state, a Cold motor start attempt has been made.
   // The time since the last Cold start attempt is accumulated.
   // The motor must confirm that it is running within RestartInhibit.Wrk_StartCheckTime minutes.
   // If it does, the state will change to S3: Cold Motor Running
   // If it does not start properly within the allowable time, the state will change to either S4: 1st Failed Cold Restart, or S5: Subsequent Cold Failed Restart.
   9: LBL(S02)OTL(Wrk_Ready);
   10: XIC(Inp_Running)CLR(Wrk_FailCount)MOV(3,Wrk_State)JMP(StartTimers);
   11: XIO(Inp_Starting)[EQU(Wrk_FailCount,1) RES(Wrk_FirstFailColdT) MOV(4,Wrk_State) ,GRT(Wrk_FailCount,1) RES(Wrk_SubsFailColdT) MOV(2,Wrk_FailCount) MOV(5,Wrk_State) ];
   12: JMP(StartTimers);
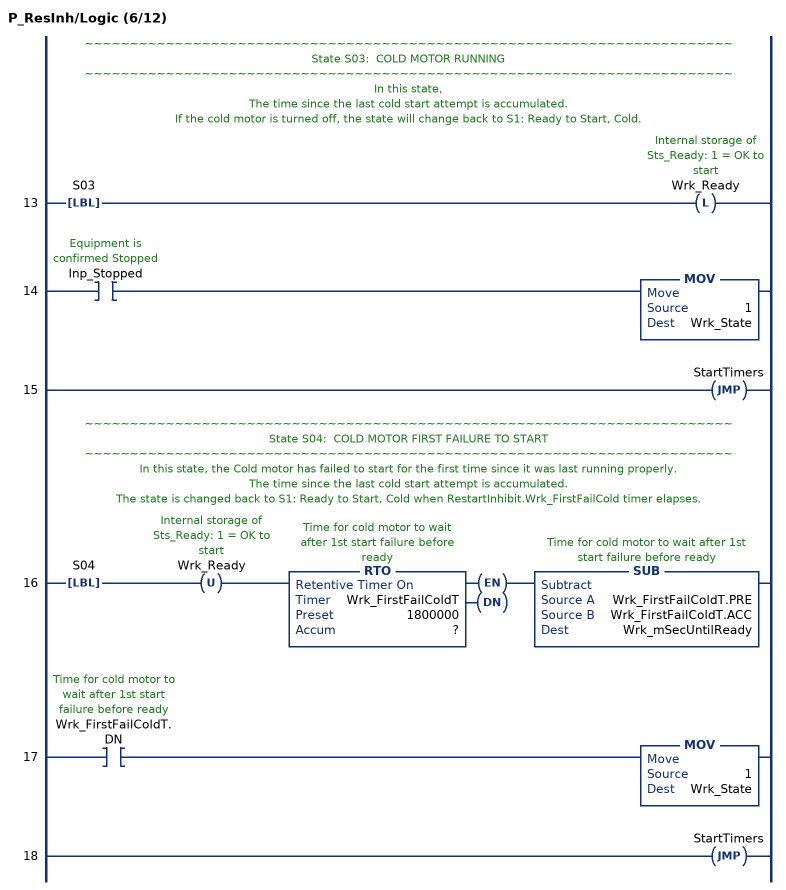
   // ~~~~~~~~~~~~~~~~~~~~~~~~~~~~~~~~~~~~~~~~~~~~~~~~~~~~~~~~~~~~~~~~~~~~~~~~
   // State S03:  COLD MOTOR RUNNING
   // ~~~~~~~~~~~~~~~~~~~~~~~~~~~~~~~~~~~~~~~~~~~~~~~~~~~~~~~~~~~~~~~~~~~~~~~~
   // In this state,
   // The time since the last cold start attempt is accumulated.
   // If the cold motor is turned off, the state will change back to S1: Ready to Start, Cold.
   13: LBL(S03)OTL(Wrk_Ready);
   14: XIC(Inp_Stopped)MOV(1,Wrk_State);
   15: JMP(StartTimers);
   // ~~~~~~~~~~~~~~~~~~~~~~~~~~~~~~~~~~~~~~~~~~~~~~~~~~~~~~~~~~~~~~~~~~~~~~~~
   // State S04:  COLD MOTOR FIRST FAILURE TO START
   // ~~~~~~~~~~~~~~~~~~~~~~~~~~~~~~~~~~~~~~~~~~~~~~~~~~~~~~~~~~~~~~~~~~~~~~~~
   // In this state, the Cold motor has failed to start for the first time since it was last running properly.
   // The time since the last cold start attempt is accumulated.
   // The state is changed back to S1: Ready to Start, Cold when RestartInhibit.Wrk_FirstFailCold timer elapses.
   16: LBL(S04)OTU(Wrk_Ready)RTO(Wrk_FirstFailColdT,?,?)SUB(Wrk_FirstFailColdT.PRE,Wrk_FirstFailColdT.ACC,Wrk_mSecUntilReady);
   17: XIC(Wrk_FirstFailColdT.DN)MOV(1,Wrk_State);
   18: JMP(StartTimers);
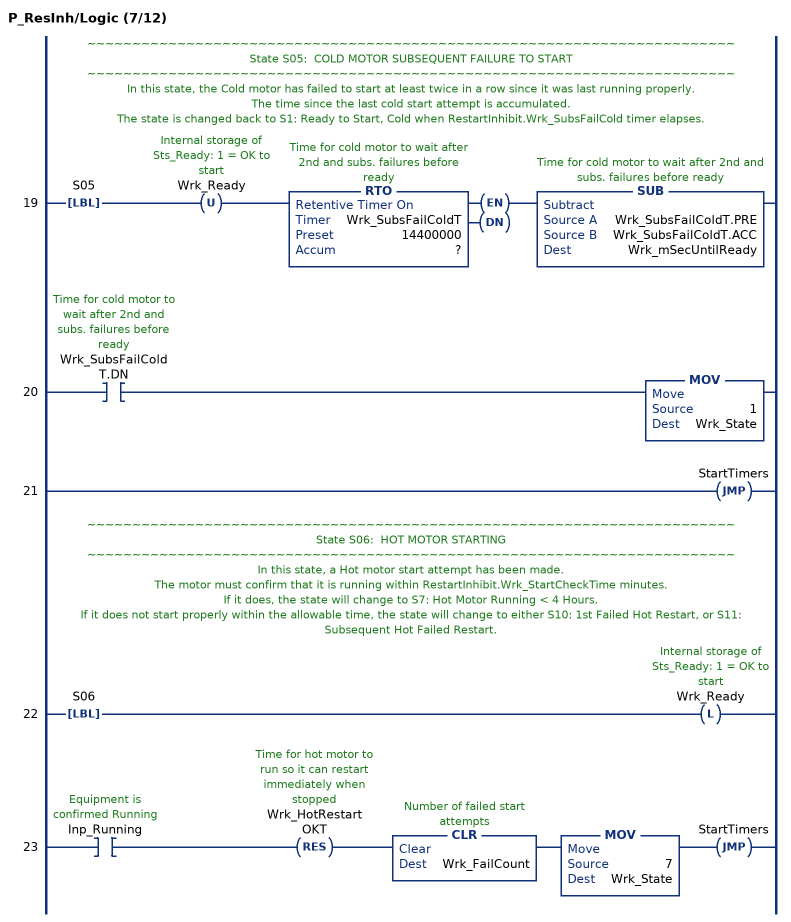
   // ~~~~~~~~~~~~~~~~~~~~~~~~~~~~~~~~~~~~~~~~~~~~~~~~~~~~~~~~~~~~~~~~~~~~~~~~
   // State S05:  COLD MOTOR SUBSEQUENT FAILURE TO START
   // ~~~~~~~~~~~~~~~~~~~~~~~~~~~~~~~~~~~~~~~~~~~~~~~~~~~~~~~~~~~~~~~~~~~~~~~~
   // In this state, the Cold motor has failed to start at least twice in a row since it was last running properly.
   // The time since the last cold start attempt is accumulated.
   // The state is changed back to S1: Ready to Start, Cold when RestartInhibit.Wrk_SubsFailCold timer elapses.
   19: LBL(S05)OTU(Wrk_Ready)RTO(Wrk_SubsFailColdT,?,?)SUB(Wrk_SubsFailColdT.PRE,Wrk_SubsFailColdT.ACC,Wrk_mSecUntilReady);
   20: XIC(Wrk_SubsFailColdT.DN)MOV(1,Wrk_State);
   21: JMP(StartTimers);
   // ~~~~~~~~~~~~~~~~~~~~~~~~~~~~~~~~~~~~~~~~~~~~~~~~~~~~~~~~~~~~~~~~~~~~~~~~
   // State S06:  HOT MOTOR STARTING
   // ~~~~~~~~~~~~~~~~~~~~~~~~~~~~~~~~~~~~~~~~~~~~~~~~~~~~~~~~~~~~~~~~~~~~~~~~
   // In this state, a Hot motor start attempt has been made.
   // The motor must confirm that it is running within RestartInhibit.Wrk_StartCheckTime minutes.
   // If it does, the state will change to S7: Hot Motor Running < 4 Hours.
   // If it does not start properly within the allowable time, the state will change to either S10: 1st Failed Hot Restart, or S11: Subsequent Hot Failed Restart.
   22: LBL(S06)OTL(Wrk_Ready);
   23: XIC(Inp_Running)RES(Wrk_HotRestartOKT)CLR(Wrk_FailCount)MOV(7,Wrk_State)JMP(StartTimers);
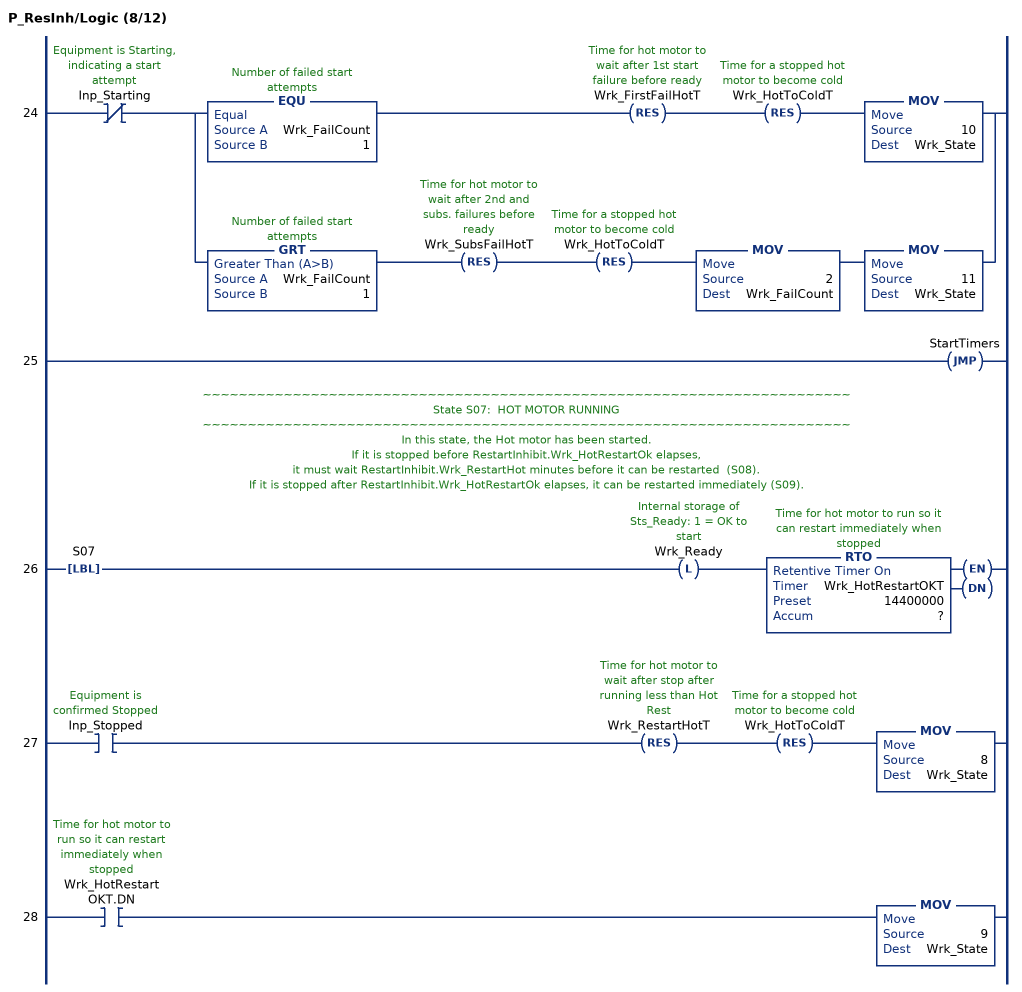
   24: XIO(Inp_Starting)[EQU(Wrk_FailCount,1) RES(Wrk_FirstFailHotT) RES(Wrk_HotToColdT) MOV(10,Wrk_State) ,GRT(Wrk_FailCount,1) RES(Wrk_SubsFailHotT) RES(Wrk_HotToColdT) MOV(2,Wrk_FailCount) MOV(11,Wrk_State) ];
   25: JMP(StartTimers);
   // ~~~~~~~~~~~~~~~~~~~~~~~~~~~~~~~~~~~~~~~~~~~~~~~~~~~~~~~~~~~~~~~~~~~~~~~~
   // State S07:  HOT MOTOR RUNNING
   // ~~~~~~~~~~~~~~~~~~~~~~~~~~~~~~~~~~~~~~~~~~~~~~~~~~~~~~~~~~~~~~~~~~~~~~~~
   // In this state, the Hot motor has been started.
   // If it is stopped before RestartInhibit.Wrk_HotRestartOk elapses,
   // it must wait RestartInhibit.Wrk_RestartHot minutes before it can be restarted  (S08).
   // If it is stopped after RestartInhibit.Wrk_HotRestartOk elapses, it can be restarted immediately (S09).
   26: LBL(S07)OTL(Wrk_Ready)RTO(Wrk_HotRestartOKT,?,?);
   27: XIC(Inp_Stopped)RES(Wrk_RestartHotT)RES(Wrk_HotToColdT)MOV(8,Wrk_State);
   28: XIC(Wrk_HotRestartOKT.DN)MOV(9,Wrk_State);
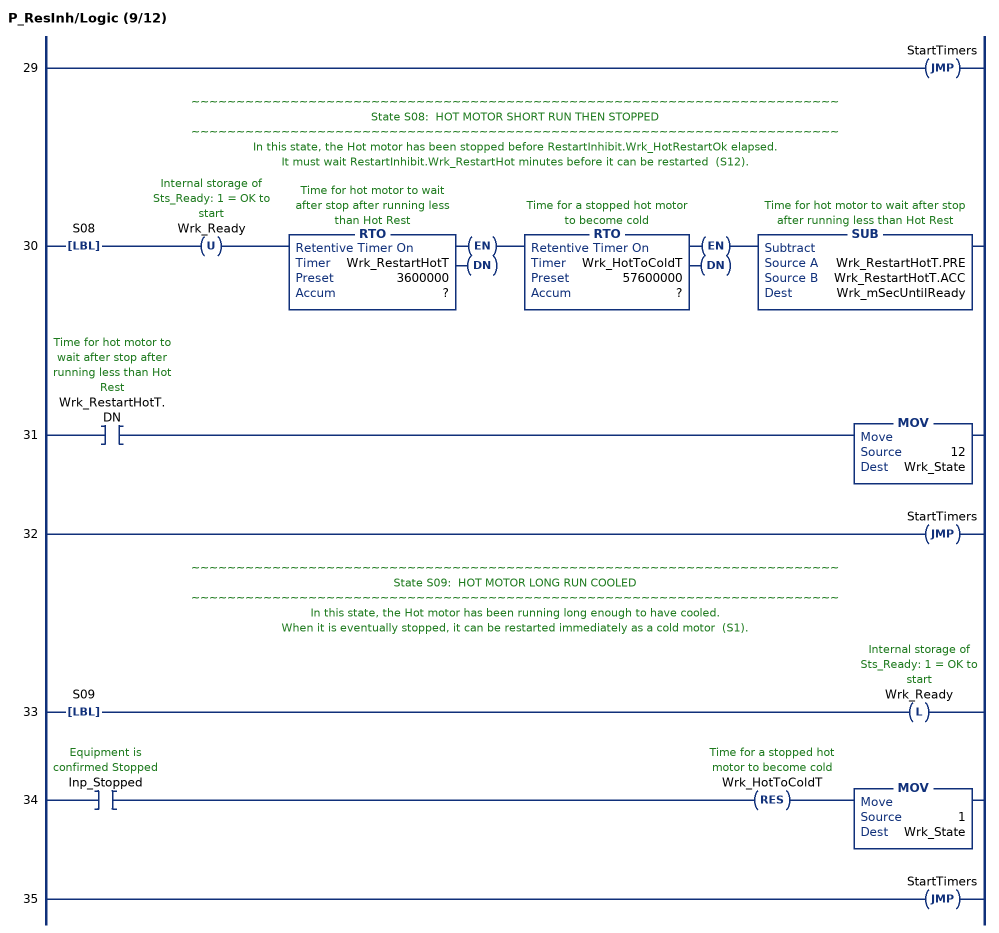
   29: JMP(StartTimers);
   // ~~~~~~~~~~~~~~~~~~~~~~~~~~~~~~~~~~~~~~~~~~~~~~~~~~~~~~~~~~~~~~~~~~~~~~~~
   // State S08:  HOT MOTOR SHORT RUN THEN STOPPED
   // ~~~~~~~~~~~~~~~~~~~~~~~~~~~~~~~~~~~~~~~~~~~~~~~~~~~~~~~~~~~~~~~~~~~~~~~~
   // In this state, the Hot motor has been stopped before RestartInhibit.Wrk_HotRestartOk elapsed.
   // It must wait RestartInhibit.Wrk_RestartHot minutes before it can be restarted  (S12).
   30: LBL(S08)OTU(Wrk_Ready)RTO(Wrk_RestartHotT,?,?)RTO(Wrk_HotToColdT,?,?)SUB(Wrk_RestartHotT.PRE,Wrk_RestartHotT.ACC,Wrk_mSecUntilReady);
   31: XIC(Wrk_RestartHotT.DN)MOV(12,Wrk_State);
   32: JMP(StartTimers);
   // ~~~~~~~~~~~~~~~~~~~~~~~~~~~~~~~~~~~~~~~~~~~~~~~~~~~~~~~~~~~~~~~~~~~~~~~~
   // State S09:  HOT MOTOR LONG RUN COOLED
   // ~~~~~~~~~~~~~~~~~~~~~~~~~~~~~~~~~~~~~~~~~~~~~~~~~~~~~~~~~~~~~~~~~~~~~~~~
   // In this state, the Hot motor has been running long enough to have cooled.
   // When it is eventually stopped, it can be restarted immediately as a cold motor  (S1).
   33: LBL(S09)OTL(Wrk_Ready);
   34: XIC(Inp_Stopped)RES(Wrk_HotToColdT)MOV(1,Wrk_State);
   35: JMP(StartTimers);
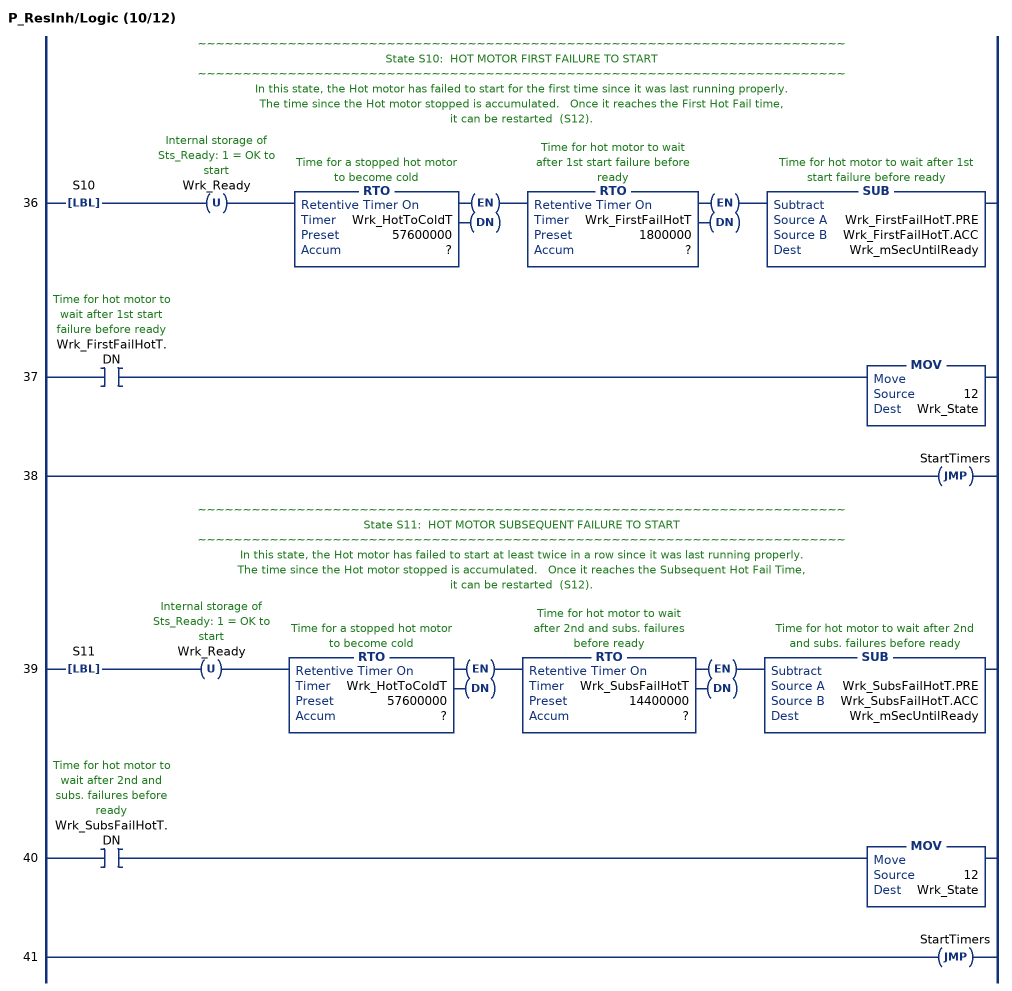
   // ~~~~~~~~~~~~~~~~~~~~~~~~~~~~~~~~~~~~~~~~~~~~~~~~~~~~~~~~~~~~~~~~~~~~~~~~
   // State S10:  HOT MOTOR FIRST FAILURE TO START
   // ~~~~~~~~~~~~~~~~~~~~~~~~~~~~~~~~~~~~~~~~~~~~~~~~~~~~~~~~~~~~~~~~~~~~~~~~
   // In this state, the Hot motor has failed to start for the first time since it was last running properly.
   // The time since the Hot motor stopped is accumulated.   Once it reaches the First Hot Fail time,
   // it can be restarted  (S12).
   36: LBL(S10)OTU(Wrk_Ready)RTO(Wrk_HotToColdT,?,?)RTO(Wrk_FirstFailHotT,?,?)SUB(Wrk_FirstFailHotT.PRE,Wrk_FirstFailHotT.ACC,Wrk_mSecUntilReady);
   37: XIC(Wrk_FirstFailHotT.DN)MOV(12,Wrk_State);
   38: JMP(StartTimers);
   // ~~~~~~~~~~~~~~~~~~~~~~~~~~~~~~~~~~~~~~~~~~~~~~~~~~~~~~~~~~~~~~~~~~~~~~~~
   // State S11:  HOT MOTOR SUBSEQUENT FAILURE TO START
   // ~~~~~~~~~~~~~~~~~~~~~~~~~~~~~~~~~~~~~~~~~~~~~~~~~~~~~~~~~~~~~~~~~~~~~~~~
   // In this state, the Hot motor has failed to start at least twice in a row since it was last running properly.
   // The time since the Hot motor stopped is accumulated.   Once it reaches the Subsequent Hot Fail Time,
   // it can be restarted  (S12).
   39: LBL(S11)OTU(Wrk_Ready)RTO(Wrk_HotToColdT,?,?)RTO(Wrk_SubsFailHotT,?,?)SUB(Wrk_SubsFailHotT.PRE,Wrk_SubsFailHotT.ACC,Wrk_mSecUntilReady);
   40: XIC(Wrk_SubsFailHotT.DN)MOV(12,Wrk_State);
   41: JMP(StartTimers);
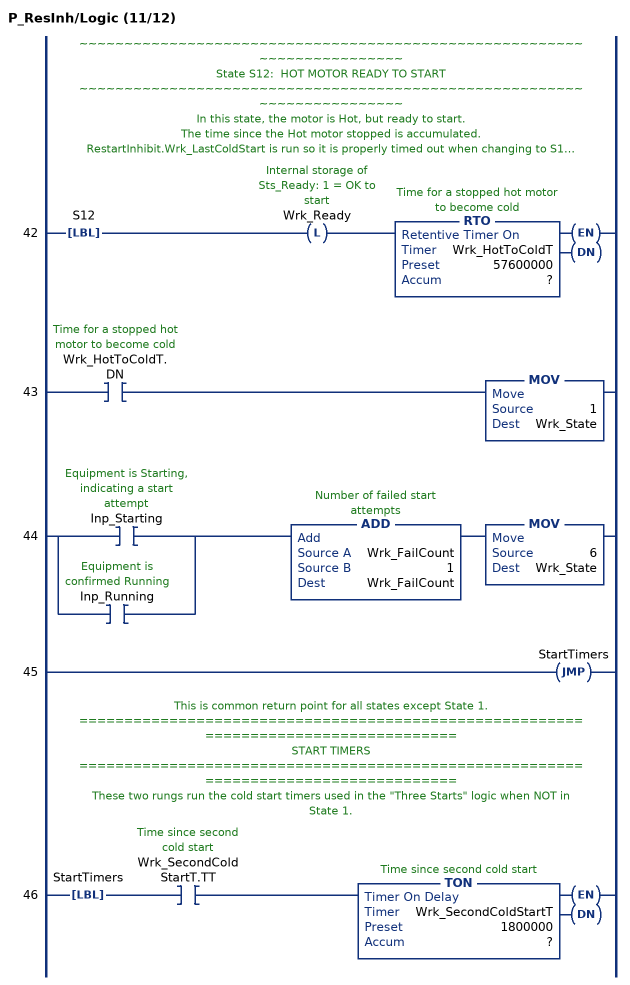
   // ~~~~~~~~~~~~~~~~~~~~~~~~~~~~~~~~~~~~~~~~~~~~~~~~~~~~~~~~~~~~~~~~~~~~~~~~
   // State S12:  HOT MOTOR READY TO START
   // ~~~~~~~~~~~~~~~~~~~~~~~~~~~~~~~~~~~~~~~~~~~~~~~~~~~~~~~~~~~~~~~~~~~~~~~~
   // In this state, the motor is Hot, but ready to start.
   // The time since the Hot motor stopped is accumulated.
   // RestartInhibit.Wrk_LastColdStart is run so it is properly timed out when changing to S1: Ready to Start, Cold.
   // If 16 hours have elapsed since the Hot motor was running, the state will be changed to S1: Ready to Start, Cold.
   // This reflects the fact that the motor has had time to cool off.
   // Otherwise, the logic waits for a Start attempt to change the state to S6: Start Check, Hot.
   42: LBL(S12)OTL(Wrk_Ready)RTO(Wrk_HotToColdT,?,?);
   43: XIC(Wrk_HotToColdT.DN)MOV(1,Wrk_State);
   44: [XIC(Inp_Starting) ,XIC(Inp_Running) ]ADD(Wrk_FailCount,1,Wrk_FailCount)MOV(6,Wrk_State);
   45: JMP(StartTimers);
   // This is common return point for all states except State 1.
   // ====================================================================================
   // START TIMERS
   // ====================================================================================
   // These two rungs run the cold start timers used in the "Three Starts" logic when NOT in State 1.
   46: LBL(StartTimers)XIC(Wrk_SecondColdStartT.TT)TON(Wrk_SecondColdStartT,?,?);
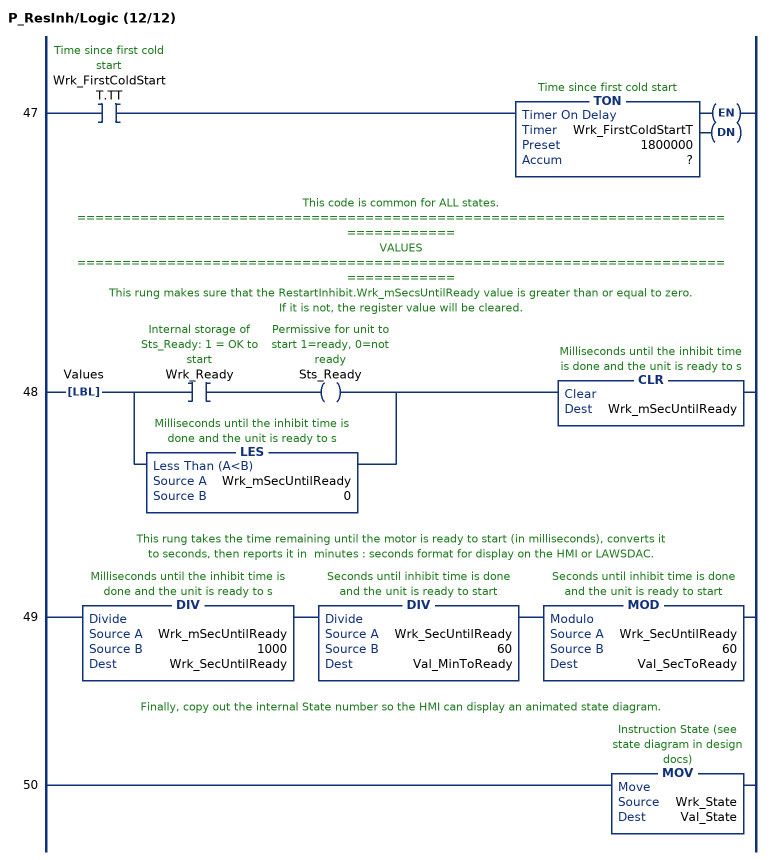
   47: XIC(Wrk_FirstColdStartT.TT)TON(Wrk_FirstColdStartT,?,?);
   // This code is common for ALL states.
   // ====================================================================================
   // VALUES
   // ====================================================================================
   // This rung makes sure that the RestartInhibit.Wrk_mSecsUntilReady value is greater than or equal to zero.
   // If it is not, the register value will be cleared.
   48: LBL(Values)[XIC(Wrk_Ready) OTE(Sts_Ready) ,LES(Wrk_mSecUntilReady,0) ]CLR(Wrk_mSecUntilReady);
   // This rung takes the time remaining until the motor is ready to start (in milliseconds), converts it
   // to seconds, then reports it in  minutes : seconds format for display on the HMI or LAWSDAC.
   49: DIV(Wrk_mSecUntilReady,1000,Wrk_SecUntilReady)DIV(Wrk_SecUntilReady,60,Val_MinToReady)MOD(Wrk_SecUntilReady,60,Val_SecToReady);
   // Finally, copy out the internal State number so the HMI can display an animated state diagram.
   50: MOV(Wrk_State,Val_State);
END_ROUTINE
